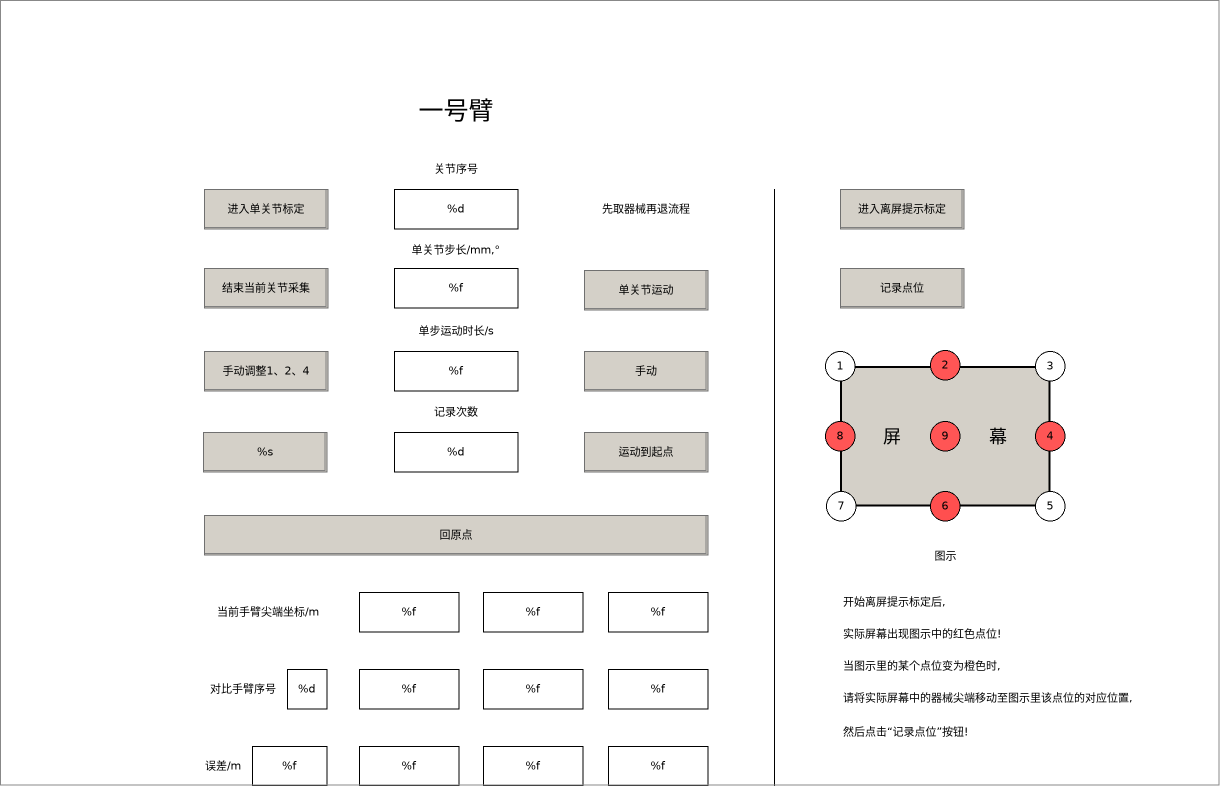
VISUALIZATION kineCali_a1  // 1220x786
    Button (204,189 124x40), "进入单关节标定", colour toggle: g_singleJntTest.m_enterSingleJntTestMode[1]
        toggle g_singleJntTest.m_enterSingleJntTestMode[1]
    Button (584,351 124x40), "手动", colour toggle: g_singleJntTest.m_manualAdjustFlag
    Button (584,432 124x40), "运动到起点", colour toggle: g_singleJntTest.m_move2StartFlag
    Rectangle (394,432 124x40), "%d", text variable: g_singleJntTest.m_dataRecordCount[1]
        OnMouseClick: write the text variable via Default, min 0, max 1000
    Label (381,230 150x40), "单关节步长/mm,°"
    Button (584,270 124x40), "单关节运动", colour toggle: g_singleJntTest.m_singleJntFlag
    Label (381,149 150x40), "关节序号"
    Rectangle (394,268 124x40), "%f", text variable: g_singleJntTest.m_jntStep
        OnMouseClick: write the text variable via Default, min 0
    Button (203,432 124x40), "%s", text variable: g_singleJntTest.m_dataRecordText, colour toggle: g_singleJntTest.m_dataRecordFlag[1]
        tap g_singleJntTest.m_dataRecordFlag[1]
    Rectangle (394,189 124x40), "%d", text variable: g_singleJntTest.m_kineCaliJntIdx
        OnMouseClick: write the text variable via Default, min 1, max 8
    Button (204,515 504x40), "回原点", colour toggle: g_singleJntTest.m_return2OriginFlag
        toggle g_singleJntTest.m_return2OriginFlag
    Rectangle (394,351 124x40), "%f", text variable: g_singleJntTest.m_EndT
        OnMouseClick: write the text variable via Default, min 0, max 100
    Label (381,311 150x40), "单步运动时长/s"
    Label (381,392 150x40), "记录次数"
    Label (394,89 124x43), "一号臂"
    Button (204,268 124x40), "结束当前关节采集", colour toggle: g_singleJntTest.m_manualEndFlag
        toggle g_singleJntTest.m_manualEndFlag
    Button (204,351 124x40), "手动调整1、2、4", colour toggle: g_singleJntTest.m_manual124StartFlag
        toggle g_singleJntTest.m_manual124StartFlag
    Label (584,189 124x40), "先取器械再退流程"
    Rectangle (359,592 100x40), "%f", text variable: g_singleJntTest.m_instruPose[1].m_pos[1]
        OnMouseClick: write the text variable via Default, min 0, max 100
    Rectangle (483,592 100x40), "%f", text variable: g_singleJntTest.m_instruPose[1].m_pos[2]
        OnMouseClick: write the text variable via Default, min 0, max 100
    Rectangle (608,592 100x40), "%f", text variable: g_singleJntTest.m_instruPose[1].m_pos[3]
        OnMouseClick: write the text variable via Default, min 0, max 100
    Rectangle (359,669 100x40), "%f", text variable: g_singleJntTest.m_instruPoseAnother.m_pos[1]
        OnMouseClick: write the text variable via Default, min 0, max 100
    Rectangle (483,669 100x40), "%f", text variable: g_singleJntTest.m_instruPoseAnother.m_pos[2]
        OnMouseClick: write the text variable via Default, min 0, max 100
    Rectangle (608,669 100x40), "%f", text variable: g_singleJntTest.m_instruPoseAnother.m_pos[3]
        OnMouseClick: write the text variable via Default, min 0, max 100
    Rectangle (287,669 40x40), "%d", text variable: g_singleJntTest.m_instruAnotherIdx
        OnMouseClick: write the text variable via Default, min 0, max 4
    Label (203,669 80x40), "对比手臂序号"
    Label (203,592 130x40), "当前手臂尖端坐标/m"
    Button (840,189 124x40), "进入离屏提示标定", colour toggle: g_offScreenTest.m_enterOffScreenTestMode[1]
        toggle g_offScreenTest.m_enterOffScreenTestMode[1]
    Line (774,189) (774,786)
    Button (840,268 124x40), "记录点位", text variable: g_singleJntTest.m_dataRecordText, colour toggle: g_offScreenTest.m_dataRecordFlag[1]
        tap g_offScreenTest.m_dataRecordFlag[1]
    Rectangle (359,746 100x40), "%f", text variable: g_singleJntTest.m_instruPoseError[1].m_pos[1]
        OnMouseClick: write the text variable via Default, min 0, max 100
    Rectangle (483,746 100x40), "%f", text variable: g_singleJntTest.m_instruPoseError[1].m_pos[2]
        OnMouseClick: write the text variable via Default, min 0, max 100
    Rectangle (608,746 100x40), "%f", text variable: g_singleJntTest.m_instruPoseError[1].m_pos[3]
        OnMouseClick: write the text variable via Default, min 0, max 100
    Rectangle (252,746 75x40), "%f", text variable: g_singleJntTest.m_instruErrDis
        OnMouseClick: write the text variable via Default, min 0, max 4
    Label (203,746 40x40), "误差/m"
    Rectangle (840,366 210x140)
    Ellipse (825,351 30x30), "1", colour toggle: g_offScreenTest.m_caliPointStartFlag[1]
        p2167032090: g_offScreenTest.m_dwAlarm
    Label (877,422 30x30), "屏"
    Label (983,422 30x30), "幕"
    Ellipse (930,350 30x30), "2", colour toggle: g_offScreenTest.m_caliPointStartFlag[2], colour variable: g_offScreenTest.m_dwNormal
        p2167032090: g_offScreenTest.m_dwAlarm
    Ellipse (1035,421 30x30), "4", colour toggle: g_offScreenTest.m_caliPointStartFlag[4], colour variable: g_offScreenTest.m_dwNormal
        p2167032090: g_offScreenTest.m_dwAlarm
    Ellipse (1035,491 30x30), "5", colour toggle: g_offScreenTest.m_caliPointStartFlag[5]
        p2167032090: g_offScreenTest.m_dwAlarm
    Ellipse (930,491 30x30), "6", colour toggle: g_offScreenTest.m_caliPointStartFlag[6], colour variable: g_offScreenTest.m_dwNormal
        p2167032090: g_offScreenTest.m_dwAlarm
    Ellipse (826,491 30x30), "7", colour toggle: g_offScreenTest.m_caliPointStartFlag[7]
        p2167032090: g_offScreenTest.m_dwAlarm
    Ellipse (825,421 30x30), "8", colour toggle: g_offScreenTest.m_caliPointStartFlag[8], colour variable: g_offScreenTest.m_dwNormal
        p2167032090: g_offScreenTest.m_dwAlarm
    Ellipse (930,421 30x30), "9", colour toggle: g_offScreenTest.m_caliPointStartFlag[9], colour variable: g_offScreenTest.m_dwNormal
        p2167032090: g_offScreenTest.m_dwAlarm
    Ellipse (1035,351 30x30), "3", colour toggle: g_offScreenTest.m_caliPointStartFlag[3]
        p2167032090: g_offScreenTest.m_dwAlarm
    Label (840,656 216x20), "当图示里的某个点位变为橙色时,"
    Label (840,688 380x20), "请将实际屏幕中的器械尖端移动至图示里该点位的对应位置,"
    Label (840,624 216x20), "实际屏幕出现图示中的红色点位!"
    Label (840,592 216x20), "开始离屏提示标定后,"
    Label (840,722 216x20), "然后点击“记录点位”按钮!"
    Label (930,546 31x20), "图示"
END_VISUALIZATION

(* stored: Version 1.1.0.1, ProductVersion 3.1.4024.11
   Visu kineCali_a1: Id {17d7edfe-a493-4318-8ea4-1046ef47c7c9} *)
